// TwinCAT 3 PLC project Untitled1
// ProgramVersion: 3.1.4024.0
// libraries:
//   Tc2_RFID, * (Beckhoff Automation GmbH)
//   Tc2_Standard, * (Beckhoff Automation GmbH)
//   Tc2_System, * (Beckhoff Automation GmbH)
//   Tc2_TcpIp, * (Beckhoff Automation GmbH)
//   Tc3_Module, * (Beckhoff Automation GmbH)
// project tree:
//   / PlcTask.TcTTO
//   POUs/ FB_System.TcPOU, FB_TcpClient.TcPOU, I_TcpClient.TcIO, MAIN.TcPOU
// real-time tasks:
//   TASK PlcTask: cycle T#10ms, priority 20, ADS port 350

CONFIGURATION Untitled1
    RESOURCE PLC ON TwinCAT3
        TASK PlcTask(INTERVAL := T#10ms, PRIORITY := 20);
        PROGRAM MAIN WITH PlcTask : MAIN;
    END_RESOURCE
END_CONFIGURATION

// ---- POUs/I_TcpClient.TcIO
INTERFACE I_TcpClient

METHOD M_Connect
VAR_INPUT
	sIP_Address : STRING;
    nPort : UINT;
END_VAR
END_METHOD

METHOD M_Cyclic
VAR_INPUT
END_VAR
END_METHOD

METHOD M_GetData : BOOL;
VAR_INPUT
	pDest : POINTER TO BYTE;
    nSize : UDINT;
END_VAR
END_METHOD

PROPERTY P_HasNewData : bool
GET
END_GET
END_PROPERTY

END_INTERFACE

// ---- POUs/MAIN.TcPOU
PROGRAM MAIN
VAR
	Hethong : FB_System;
END_VAR

Hethong();

END_PROGRAM

// ---- POUs/FB_System.TcPOU
FUNCTION_BLOCK FB_System
VAR_INPUT
END_VAR
VAR_OUTPUT
END_VAR
VAR
	fbTcpTest    : FB_TcpClient;
    bStartTest   : BOOL;
    arrDataRx    : ARRAY[0..255] OF BYTE;
END_VAR

// Kích hoạt kết nối thử nghiệm
IF bStartTest THEN
    fbTcpTest.M_Connect(sIP_Address := '192.168.1.190', nPort := 6000);
    bStartTest := FALSE;
END_IF

// Gọi trái tim động cơ chạy liên tục
fbTcpTest.M_Cyclic();

// Hứng dữ liệu test
IF fbTcpTest.P_HasNewData THEN
    fbTcpTest.M_GetData(pDest := ADR(arrDataRx), nSize := SIZEOF(arrDataRx));
END_IF

END_FUNCTION_BLOCK

// ---- POUs/FB_TcpClient.TcPOU
FUNCTION_BLOCK FB_TcpClient IMPLEMENTS I_TcpClient
VAR_INPUT
END_VAR
VAR_OUTPUT
END_VAR
VAR
	fbConnect    : FB_SocketConnect;
    fbReceive    : FB_SocketReceive;
    hSocket      : T_HSOCKET;
    nState       : INT := 0;
    
    // Vùng nhớ đệm mạng
    arrBuffer    : ARRAY[0..255] OF BYTE;
    bDataReady   : BOOL := FALSE;
    
    // Biến lưu IP và Port từ Method truyền vào
    sTargetIP    : STRING;
    nTargetPort  : UINT;
    bCmdConnect  : BOOL;
END_VAR

{warning 'add method implementation '}
METHOD M_Connect
VAR_INPUT
	sIP_Address	: STRING;
	nPort	: UINT;
END_VAR
sTargetIP := sIP_Address;
nTargetPort := nPort;
bCmdConnect := TRUE; // Bóp cò để M_Cyclic bắt đầu chạy
END_METHOD

{warning 'add method implementation '}
METHOD M_Cyclic
// Gọi các khối hàm hệ thống ở đầu Method
fbConnect();
fbReceive();

CASE nState OF
    0: // CHỜ KẾT NỐI
        IF bCmdConnect THEN
            bCmdConnect := FALSE;
            nState := 10;
        END_IF

    10: // GỌI HÀM KẾT NỐI (Logic y hệt như cũ)
        fbConnect.sRemoteHost := sTargetIP;
        fbConnect.nRemotePort := nTargetPort;
        fbConnect.bExecute := TRUE;
        // ... (các đoạn check bBusy, bError giữ nguyên)

    20: // LẮNG NGHE DỮ LIỆU
        fbReceive.hSocket := hSocket;
        fbReceive.cbLen := SIZEOF(arrBuffer);
        fbReceive.pDest := ADR(arrBuffer);
        fbReceive.bExecute := TRUE;
        // ... (check nRecBytes > 0 rồi bật cờ bDataReady)
END_CASE
END_METHOD

{warning 'add method implementation '}
METHOD M_GetData : BOOL;
VAR_INPUT
	pDest	: POINTER TO BYTE;
	nSize	: UDINT;
END_VAR
IF bDataReady THEN
    MEMCPY(destAddr := pDest, srcAddr := ADR(arrBuffer), n := nSize);
    bDataReady := FALSE; // Reset cờ sau khi đã lấy xong
    M_GetData := TRUE;
ELSE
    M_GetData := FALSE;
END_IF
END_METHOD

{warning 'add property implementation'}
PROPERTY P_HasNewData : BOOL
GET
P_HasNewData := bDataReady;
END_GET
END_PROPERTY

END_FUNCTION_BLOCK
